// Mitsubishi GX Works2 project: tutor06_modbustcp_ladder   PLC: FX1N/FX1NC

PROGRAM MAIN
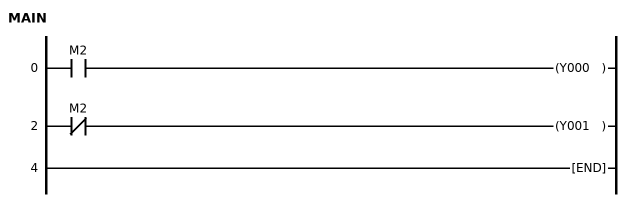
0     LD      M2
      OUT     Y000
2     LDI     M2
      OUT     Y001
4     END
END_PROGRAM
